FUNCTION_BLOCK FB_Arm
VAR
	bActivated			: BOOL;
	bBusy				: BOOL;
	bRunning			: BOOL;
	bLoad				: BOOL;
	bUnload				: BOOL;
	
	rCurX				: REAL;
	rCurY				: REAL;
	
	rImportX			: REAL;
	rExportX			: REAL;
	rLoadingY			: REAL	:= 0;
	
	rIdleX				: REAL	:= 0;
	rIdleY				: REAL	:= 10;
	
	stUnit				: ST_Unit;
	
	iType				: INT;
	iCase				: INT;
END_VAR

PROPERTY Activated : BOOL
GET
Activated := bActivated;
END_GET
SET
bActivated := Activated;
END_SET
END_PROPERTY

METHOD Assign : PVOID
VAR_INPUT
	ImportLocation			: REAL;
	ExportLocation			: REAL;
	UnitType				: INT;
END_VAR
IF NOT bBusy AND bActivated THEN
	bBusy := TRUE;
	rImportX := ImportLocation;
	rExportX := ExportLocation;
	iType := UnitType;
END_IF
END_METHOD

PROPERTY Busy : BOOL
GET
Busy := bBusy;
END_GET
END_PROPERTY

PROPERTY CurUnit : ST_Unit
GET
CurUnit := stUnit;
stUnit.eType := -1;
END_GET
SET
IF CurUnit.eType <> -1 THEN
	stUnit := CurUnit;
END_IF
END_SET
END_PROPERTY

PROPERTY CurX : REAL
GET
CurX := rCurX;
END_GET
SET
rCurX := CurX;
END_SET
END_PROPERTY

PROPERTY CurY : REAL
GET
CurY := rCurY;
END_GET
SET
rCurY := CurY;
END_SET
END_PROPERTY

PROPERTY Load : BOOL
GET
Load := bLoad;
END_GET
SET
bLoad := Load;
END_SET
END_PROPERTY

METHOD Run : PVOID
VAR_INPUT
END_VAR
IF NOT bBusy THEN
	iCase := 0;
END_IF
IF bBusy AND NOT bRunning THEN
	bRunning := TRUE;
	iCase := 1;
END_IF

CASE iCase OF
	0:	(*Idle*)
		IF rCurY < rIdleY THEN
			rCurY := rCurY + 1;
		ELSIF
			rCurY > rIdleY THEN
			rCurY := rCurY - 1;
		ELSE
			IF rCurX < rIdleX THEN
				rCurX := rCurX + 1;
			ELSIF 
				rCurX > rIdleX THEN
				rCurX := rCurX - 1;
			END_IF
		END_IF
		
	1:	(*Go Import Location*)
		IF rCurY < rIdleY THEN
			rCurY := rCurY + 1;
		ELSIF
			rCurY > rIdleY THEN
			rCurY := rCurY - 1;
		ELSE
			IF rCurX < rImportX THEN
				rCurX := rCurX + 1;
			ELSIF
				rCurX > rImportX THEN
				rCurX := rCurX - 1;
			ELSE
				iCase := 11;
			END_IF
		END_IF
		
	11:	(*Go to Loading Position*)
		IF rCurY < rLoadingY THEN
			rCurY := rCurY + 1;
		ELSIF 
			rCurY > rLoadingY THEN
			rCurY := rCurY - 1;
		ELSE
			bLoad := TRUE;
			iCase := 2;
		END_IF
	
	2:	(*Load*)
		IF NOT bLoad THEN
			iCase := 3;
		END_IF
		
	21:	(*Leave Loading Position*)
		IF rCurY < rIdleY THEN
			rCurY := rCurY + 1;
		ELSIF
			rCurY > rIdleY THEN
			rCurY := rCurY - 1;
		ELSE
			iCase := 3;
		END_IF
	
	3:	(*Go to Export Location*)
		IF rCurX < rExportX THEN
			rCurX := rCurX + 1;
		ELSIF
			rCurX > rExportX THEN
			rCurX := rCurX - 1;
		ELSE
			IF rCurY < rLoadingY THEN
				rCurY := rCurY + 1;
			ELSIF 
				rCurY > rLoadingY THEN
				rCurY := rCurY - 1;
			ELSE
				bUnload := TRUE;
				iCase := 4;
			END_IF
		END_IF
		
	4:	(*Unload*)
		IF NOT bUnload THEN
			iCase := 0;
			bBusy := FALSE;
			bRunning := FALSE;
		END_IF
	
END_CASE
END_METHOD

PROPERTY UnitType : INT
GET
UnitType := iType;
END_GET
END_PROPERTY

PROPERTY Unload : BOOL
GET
Unload := bUnload;
END_GET
SET
bUnload := Unload;
END_SET
END_PROPERTY

END_FUNCTION_BLOCK

(* stored: Version 1.1.0.1, ProductVersion 3.1.4024.12
   POU FB_Arm: Id {75e5cc7f-f676-4e64-a36d-5261779273ee}, SpecialFunc None
   Folder Properties: Id {25cccf8b-0fa1-49ed-8a26-204ec71a3376}
   Property Activated: Id {b0b6577a-e8c5-4910-a542-0354fbd42b1b}
   Get Get: Id {b0c904f5-fe06-4484-845d-0ce3e10cc3f7}
   Set Set: Id {939fe8cd-62b3-40d3-bf60-5f2504838f18}
   Method Assign: Id {9bb5c29b-9d76-4d01-97cf-5478495eb455}
   Property Busy: Id {8c5ac7e7-f0c0-4896-b082-5b2313de9b57}
   Get Get: Id {68774231-fe23-406b-bd03-1efb75470149}
   Property CurUnit: Id {1899013a-b7fc-4670-aff4-000bfd1ad739}
   Get Get: Id {c5762c6d-71ea-472b-9f5e-1e86bf3f481b}
   Set Set: Id {30092054-f23c-456f-9e34-f94309ebb517}
   Property CurX: Id {d472d742-8be1-43bd-813c-52ab9aa89f69}
   Get Get: Id {ad840bed-414e-4564-8b17-16b99a530ca0}
   Set Set: Id {19af05a2-01e6-41b0-a3f4-323a1f0e6444}
   Property CurY: Id {03d3888b-82e5-4e76-85ce-b464b921a7a4}
   Get Get: Id {bdfea8e1-9a3c-4656-a882-a51b3e90b23d}
   Set Set: Id {8cae0b24-30f7-4439-a422-c3b8936e8664}
   Property Load: Id {8fc9fcc9-9d21-4577-8b11-ab846c03ffec}
   Get Get: Id {c558f3cc-da82-45cb-96ba-d8cece26a63f}
   Set Set: Id {1435226d-2278-4a45-81e8-550a8aeff9ba}
   Method Run: Id {dbae01e7-931c-4469-a7fb-490b8d311ea3}
   Property UnitType: Id {b77ae1b4-93f7-4341-adb3-d352fd9e7bd0}
   Get Get: Id {fabec5dd-a5f6-408c-bef5-b9fe95971027}
   Property Unload: Id {11071653-373e-41a3-8cbb-ac2a93b8c962}
   Get Get: Id {4af0a6a7-95d3-433d-8b2e-58bc42e700c8}
   Set Set: Id {e78288a0-5f10-4323-afde-a4919b0e56f4} *)
